// Passes in one scan. The baseline for suite-level counting.

//

// Records a check deliberately: a body that checks nothing is reported Errored,

// not Passed, so a double that asserted nothing would quietly test the wrong

// thing.
FUNCTION_BLOCK PassingTest IMPLEMENTS I_Test
VAR
	_BodyCalls : UDINT;
END_VAR

// How many times a suite has run this. A re-run doubles it; an individual re-run

// raises it without touching any count the suite reports.
PROPERTY BodyCalls : UDINT
GET
BodyCalls := _BodyCalls;
END_GET
END_PROPERTY

METHOD Run : BOOL
VAR_INPUT
	Enable : BOOL;
	Test   : I_TestAssertions;
END_VAR
IF NOT Enable THEN
	Run := TRUE;
	RETURN;
END_IF

_BodyCalls := _BodyCalls + 1;
Test.AssertTrue(TRUE, 'this one passes');
Run := TRUE;
END_METHOD

END_FUNCTION_BLOCK

(* stored: Version 1.1.0.1, ProductVersion 3.1.4026.18
   POU PassingTest: Id {2525e98b-0b5d-457d-9df3-dee4e022981e}, SpecialFunc None
   Folder I_Test: Id {db3f0779-dab9-4ee1-b1a2-75d871e7af76}
   Property BodyCalls: Id {c49ae0e5-6334-4810-88dd-9e1cb6811a5d}
   Get Get: Id {338b3530-0ba7-4790-bf90-ee8b762563bf}
   Method Run: Id {659503aa-96e3-4305-866b-9b269b49e360} *)
